ABB RAPID module: 000DE578

MODULE Module1
	CONST robtarget PickLeft:=[[360.5,88.055,133.879],[0,1,0,0],[-1,0,-1,0],[9E+09,9E+09,9E+09,9E+09,9E+09,9E+09]];
	CONST robtarget HomeLeft:=[[477.5,-145.945,302.406],[0,1,0,0],[0,0,0,0],[9E+09,9E+09,9E+09,9E+09,9E+09,9E+09]];
	CONST robtarget Left11:=[[415.5,-515.945,197.406],[0,1,0,0],[0,0,0,0],[9E+09,9E+09,9E+09,9E+09,9E+09,9E+09]];
	CONST robtarget Left12:=[[415.5,-625.945,197.406],[0,1,0,0],[0,0,0,0],[9E+09,9E+09,9E+09,9E+09,9E+09,9E+09]];
	CONST robtarget Left21:=[[415.5,-515.945,302.406],[0,1,0,0],[0,0,0,0],[9E+09,9E+09,9E+09,9E+09,9E+09,9E+09]];
	CONST robtarget Left22:=[[415.5,-625.945,302.406],[0,1,0,0],[0,0,0,0],[9E+09,9E+09,9E+09,9E+09,9E+09,9E+09]];
    !***********************************************************
    !
    ! Module:  Left Stacker robot
    !
    ! Description:
    !   <Insert description here>
    !
    ! Author: madsw
    ! Version: 1.0
    !
    !***********************************************************
    PROC main()
        !Add your code here
    ENDPROC
ENDMODULE
